# EPICS substitutions: db/amo.substitutions
file "ecmcEcSlave.template"
{
  pattern {}
          {}
}

# All fields related to postion scaling and alarms
file "ecmcEL5021-chX.template"
{
  pattern {CH_ID, LINR,    ESLO,                  EOFF,   EGU,        PREC, LOW, LOLO, HIGH, HIHI, HYST, LLSV,       LSV,        HSV,        HHSV      }
          {01,    "SLOPE", 0.00017166137695,      0,      "Deg",    0,    0,   0,    0,    0,    0,    "NO_ALARM", "NO_ALARM", "NO_ALARM", "NO_ALARM"}
}
